// TIA Portal V20 export
FUNCTION "StepToString" : String   // FC90, SCL
// stored: Namespace Unit1.Em4, SetENOAutomatically false
   VAR_INPUT
      StepDINT : DInt;   // DINT value of the step
   END_VAR
BEGIN
   // Translates the sequence step number to the step name
   // Adjusted for Sequence_1_Cutter real use case

   CASE #StepDINT OF
       1:
           #StepToString := 'Idle';

       101:
           #StepToString := 'JOB[1] Condition';
       111:
           #StepToString := 'Axis Homed Check';
       121:
           #StepToString := 'Axis HomePos Check';
       131:
           #StepToString := 'Feeding Cylinder WorkPos Check';
       191:
           #StepToString := 'JOB[1] Step End';

       901:
           #StepToString := 'Immediate Stop';

       ELSE
           #StepToString := 'N/A';

   END_CASE;
END_FUNCTION
